(* IEC 61131-3 sources: eCockpitGit/test_project/src/%F%00 Library/%F%Common Functions/%F%Linearsation/%F%BYTE, 4 files *)

(* ---- %POU%FU_bLinear2.st ---- *)
//This function, converts an x, value to an y value using and 2 points on the x and y scale
// +-----------+----------+----------+-----------------------------------------------------------------------------------------------------------------------+
// |**Version**|**Author**| **Date** |**Changes**                                                                                                            |
// +-----------+----------+----------+-----------------------------------------------------------------------------------------------------------------------+
// | 1         | NSN      | 21-06-18 | Creation                                                                                                              |
// +-----------+----------+----------+-----------------------------------------------------------------------------------------------------------------------+
FUNCTION FU_bLinear2 : BYTE
VAR_INPUT
	XIn		:BYTE;
	X1		:BYTE;
	X2		:BYTE;
	Y1		:BYTE;
	Y2		:BYTE;
END_VAR
VAR
	a		:REAL;
	b		:REAL;
END_VAR
(*%!%__DELIMITER__%!%*)
IF X2 > X1 THEN
	//a value is calculated
	IF X2 - X1 = 0 THEN	a := 0; ELSE a := TO_REAL((Y2 - Y1)) / (X2 - X1); END_IF
	//b value is calculated
	b 							:=		TO_REAL(Y1) - (a * TO_REAL(X1));
	//Output is calculated
	FU_bLinear2 				:=		TO_BYTE(a * TO_REAL (XIn) + b);
ELSE
	//a value is calculated
	IF X2 - X1 = 0 THEN	a := 0; ELSE a := TO_REAL((Y2 - Y1)) / (X2 - X1); END_IF
	//b value is calculated
	b 							:=		TO_REAL(Y1) - (a * TO_REAL(X1));
	//Output is calculated
	FU_bLinear2 				:=		TO_BYTE(a * TO_REAL (XIn) + b);
END_IF

(* ---- %POU%FU_bLinear2Ends.st ---- *)
//This function, converts an x, value to an y value using and 2 points on the x and y scale
//This function has ends, which means the output is never greater or smaller than the range of y
// +-----------+----------+----------+-----------------------------------------------------------------------------------------------------------------------+
// |**Version**|**Author**| **Date** |**Changes**                                                                                                            |
// +-----------+----------+----------+-----------------------------------------------------------------------------------------------------------------------+
// | 1         | NSN      | 21-06-18 | Creation                                                                                                              |
// +-----------+----------+----------+-----------------------------------------------------------------------------------------------------------------------+
FUNCTION FU_bLinear2Ends : BYTE
VAR_INPUT
	XIn		:BYTE;
	X1		:BYTE;
	X2		:BYTE;
	Y1		:BYTE;
	Y2		:BYTE;
END_VAR
VAR
	a		:REAL;
	b		:REAL;
END_VAR
(*%!%__DELIMITER__%!%*)
IF X2 > X1 THEN
	IF XIn <= X1 THEN	//When input is out of bounds
		FU_bLinear2Ends 			:=		Y1;
	ELSIF XIn >= X2 THEN	//When input is out of bounds
		FU_bLinear2Ends 			:=		Y2;
	ELSIF XIn > X1 AND XIn < X2 THEN	//When input is with the
		//a value is calculated
		IF X2 - X1 = 0 THEN	a := 0; ELSE a := TO_REAL((Y2 - Y1)) / (X2 - X1); END_IF
		//b value is calculated
		b 							:=		TO_REAL(Y1) - (a * TO_REAL(X1));
		//Output is calculated
		FU_bLinear2Ends 			:=		TO_BYTE(a * TO_REAL (XIn) + b);
	END_IF
ELSE
	IF XIn >= X1 THEN
		FU_bLinear2Ends 			:=		Y1;
	ELSIF XIn <= X2 THEN
		FU_bLinear2Ends 			:=		Y2;
	ELSIF XIn < X1 AND XIn > X2 THEN
		//a value is calculated
		IF X2 - X1 = 0 THEN	a := 0; ELSE a := TO_REAL((Y2 - Y1)) / (X2 - X1); END_IF
		//b value is calculated
		b 							:=		TO_REAL(Y1) - (a * TO_REAL(X1));
		//Output is calculated
		FU_bLinear2Ends 			:=		TO_BYTE(a * TO_REAL (XIn) + b);
	END_IF
END_IF

(* ---- %POU%FU_bLinear3Ends.st ---- *)
//This function, converts an x, value to an y value using and 3 points on the x and y scale
//This function has ends, which means the output is never greater or smaller than the range of y
// +-----------+----------+----------+-----------------------------------------------------------------------------------------------------------------------+
// |**Version**|**Author**| **Date** |**Changes**                                                                                                            |
// +-----------+----------+----------+-----------------------------------------------------------------------------------------------------------------------+
// | 1         | NSN      | 10-01-18 | Updated to new format                                                                                                 |
// +-----------+----------+----------+-----------------------------------------------------------------------------------------------------------------------+
// | 1         | NSN      | 13-06-18 | Updated names and types                                                                                               |
// +-----------+----------+----------+-----------------------------------------------------------------------------------------------------------------------+
FUNCTION FU_bLinear3Ends : BYTE
VAR_INPUT
	XIn		:BYTE;
	X1		:BYTE;
	X2		:BYTE;
	X3		:BYTE;
	Y1		:BYTE;
	Y2		:BYTE;
	Y3		:BYTE;
END_VAR
VAR
	a		:REAL;
	b		:REAL;
END_VAR
(*%!%__DELIMITER__%!%*)
IF X3 > X1 THEN
	IF XIn <= X1 THEN	//When input is out of bounds
		FU_bLinear3Ends 			:=		Y1;
	ELSIF XIn >= X3 THEN	//When input is out of bounds
		FU_bLinear3Ends 			:=		Y3;
	ELSIF XIn > X1 AND XIn <= X2 THEN	//When input is with the
		//a value is calculated
		IF X2 - X1 = 0 THEN	a := 0; ELSE a := TO_REAL((Y2 - Y1)) / (X2 - X1); END_IF
		//b value is calculated
		b 							:=		TO_REAL(Y1) - (a * TO_REAL(X1));
		//Output is calculated
		FU_bLinear3Ends 			:=		TO_BYTE(a * TO_REAL (XIn) + b);
	ELSIF XIn > X2 AND XIn < X3 THEN
		//a value is calculated
		IF X3 - X2 = 0 THEN	a := 0; ELSE a := TO_REAL((Y3 - Y2)) / (X3 - X2); END_IF
		//b value is calculated
		b 							:=		TO_REAL(Y2) - (a * TO_REAL(X2));
		//Output is calculated
		FU_bLinear3Ends 			:=		TO_BYTE(a * TO_REAL (XIn) + b);
	END_IF
ELSE
	IF XIn >= X1 THEN
		FU_bLinear3Ends 			:=		Y1;
	ELSIF XIn <= X3 THEN
		FU_bLinear3Ends 			:=		Y3;
	ELSIF XIn < X1 AND XIn >= X2 THEN
		//a value is calculated
		IF X2 - X1 = 0 THEN	a := 0; ELSE a := TO_REAL((Y2 - Y1)) / (X2 - X1); END_IF
		//b value is calculated
		b 							:=		TO_REAL(Y1) - (a * TO_REAL(X1));
		//Output is calculated
		FU_bLinear3Ends 			:=		TO_BYTE(a * TO_REAL (XIn) + b);
	ELSIF XIn < X2 AND XIn > X3 THEN
		//a value is calculated
		IF X3 - X2 = 0 THEN	a := 0; ELSE a := TO_REAL((Y3 - Y2)) / (X3 - X2); END_IF
		//b value is calculated
		b 							:=		TO_REAL(Y2) - (a * TO_REAL(X2));
		//Output is calculated
		FU_bLinear3Ends 			:=		TO_BYTE(a * TO_REAL (XIn) + b);
	END_IF
END_IF

(* ---- %POU%FU_bLinear4Ends.st ---- *)
//This function, converts an x, value to an y value using and 3 points on the x and y scale
//This function has ends, which means the output is never greater or smaller than the range of y
// +-----------+----------+----------+-----------------------------------------------------------------------------------------------------------------------+
// |**Version**|**Author**| **Date** |**Changes**                                                                                                            |
// +-----------+----------+----------+-----------------------------------------------------------------------------------------------------------------------+
// | 1         | NSN      | 30-05-18 | Updated to new format                                                                                                 |
// +-----------+----------+----------+-----------------------------------------------------------------------------------------------------------------------+
FUNCTION FU_bLinear4Ends : BYTE
VAR_INPUT
	XIn		:BYTE;
	X1		:BYTE;
	X2		:BYTE;
	X3		:BYTE;
	X4		:BYTE;
	Y1		:BYTE;
	Y2		:BYTE;
	Y3		:BYTE;
	Y4		:BYTE;
END_VAR
VAR
	a		:REAL;
	b		:REAL;
END_VAR
(*%!%__DELIMITER__%!%*)
IF X4 > X1 THEN
	IF XIn <= X1 THEN	//When input is out of bounds
		FU_bLinear4Ends 			:=		Y1;
	ELSIF XIn >= X4 THEN	//When input is out of bounds
		FU_bLinear4Ends 			:=		Y4;
	ELSIF XIn > X1 AND XIn <= X2 THEN	//When input is with the
		//a value is calculated
		IF X2 - X1 = 0 THEN	a := 0; ELSE a := TO_REAL((Y2 - Y1)) / (X2 - X1); END_IF
		//b value is calculated
		b 							:=		TO_REAL(Y1) - (a * TO_REAL(X1));
		//Output is calculated
		FU_bLinear4Ends 			:=		TO_BYTE(a * TO_REAL (XIn) + b);
	ELSIF XIn > X2 AND XIn <= X3 THEN
		//a value is calculated
		IF X3 - X2 = 0 THEN	a := 0; ELSE a := TO_REAL((Y3 - Y2)) / (X3 - X2); END_IF
		//b value is calculated
		b 							:=		TO_REAL(Y2) - (a * TO_REAL(X2));
		//Output is calculated
		FU_bLinear4Ends 			:=		TO_BYTE(a * TO_REAL (XIn) + b);
	ELSIF XIn > X3 AND XIn < X4 THEN
		//a value is calculated
		IF X4 - X3 = 0 THEN	a := 0; ELSE a := TO_REAL((Y4 - Y3)) / (X4 - X3); END_IF
		//b value is calculated
		b 							:=		TO_REAL(Y3) - (a * TO_REAL(X3));
		//Output is calculated
		FU_bLinear4Ends 			:=		TO_BYTE(a * TO_REAL (XIn) + b);
	END_IF
ELSE
	IF XIn >= X1 THEN
		FU_bLinear4Ends 			:=		Y1;
	ELSIF XIn <= X4 THEN
		FU_bLinear4Ends 			:=		Y4;
	ELSIF XIn < X1 AND XIn >= X2 THEN
		//a value is calculated
		IF X2 - X1 = 0 THEN	a := 0; ELSE a := TO_REAL((Y2 - Y1)) / (X2 - X1); END_IF
		//b value is calculated
		b 							:=		TO_REAL(Y1) - (a * TO_REAL(X1));
		//Output is calculated
		FU_bLinear4Ends 			:=		TO_BYTE(a * TO_REAL (XIn) + b);
	ELSIF XIn < X2 AND XIn >= X3 THEN
		//a value is calculated
		IF X3 - X2 = 0 THEN	a := 0; ELSE a := TO_REAL((Y3 - Y2)) / (X3 - X2); END_IF
		//b value is calculated
		b 							:=		TO_REAL(Y2) - (a * TO_REAL(X2));
		//Output is calculated
		FU_bLinear4Ends 			:=		TO_BYTE(a * TO_REAL (XIn) + b);
	ELSIF XIn < X3 AND XIn > X4 THEN
		//a value is calculated
		IF X4 - X3 = 0 THEN	a := 0; ELSE a := TO_REAL((Y4 - Y3)) / (X4 - X3); END_IF
		//b value is calculated
		b 							:=		TO_REAL(Y3) - (a * TO_REAL(X3));
		//Output is calculated
		FU_bLinear4Ends 			:=		TO_BYTE(a * TO_REAL (XIn) + b);
	END_IF
END_IF
